// SYNTAX TEST "Step7 AWL.sublime-syntax"

// ==================================================
//  common
//  Performance: 3.0ms
// ==================================================

///////////////////////////////////////////////////////////////////////////////
// namespaces                                                                //
///////////////////////////////////////////////////////////////////////////////

NAMESPACE Name
// <- meta.namespace.plc keyword.declaration.namespace.begin.plc
//^^^^^^^^^^^^^ meta.namespace.plc
//^^^^^^^ keyword.declaration.namespace.begin.plc
//        ^^^^ entity.name.namespace.plc
//            ^ meta.fold.namespace.begin.plc
    TYPE
//  ^^^^^ meta.namespace.plc meta.block.udt.header.plc
//  ^^^^ keyword.declaration.udt.begin.plc
    END_TYPE
//  ^^^^^^^^ meta.namespace.plc keyword.declaration.udt.end.plc

    DATA_BLOCK "dataBlock"
//  ^^^^^^^^^^^^^^^^^^^^^^ meta.namespace.plc meta.block.db.header.plc
//  ^^^^^^^^^^ keyword.declaration.db.begin.plc
//             ^^^^^^^^^^^ entity.name.datablock.plc
//             ^ punctuation.definition.variable.begin.plc
//                       ^ punctuation.definition.variable.end.plc
    END_DATA_BLOCK
//  ^^^^^^^^^^^^^^ meta.namespace.plc keyword.declaration.db.end.plc

    FUNCTION_BLOCK "funcName"
//  ^^^^^^^^^^^^^^^^^^^^^^^^^ meta.namespace.plc meta.block.fb.header.plc
//  ^^^^^^^^^^^^^^ keyword.declaration.fb.begin.plc
//                 ^^^^^^^^^^ entity.name.function.plc
//                 ^ punctuation.definition.variable.begin.plc
//                          ^ punctuation.definition.variable.end.plc
    END_FUNCTION_BLOCK
//  ^^^^^^^^^^^^^^^^^^ meta.namespace.plc keyword.declaration.fb.end.plc

    FUNCTION "funcName"
//  ^^^^^^^^^^^^^^^^^^^ meta.namespace.plc meta.block.fc.header.plc
//  ^^^^^^^^ keyword.declaration.fc.begin.plc
//           ^^^^^^^^^^ entity.name.function.plc
//           ^ punctuation.definition.variable.begin.plc
//                    ^ punctuation.definition.variable.end.plc
    END_FUNCTION
//  ^^^^^^^^^^^^ meta.namespace.plc keyword.declaration.fc.end.plc

    ORGANIZATION_BLOCK "BlockName"
//  ^^^^^^^^^^^^^^^^^^^^^^^^^^^^^^ meta.namespace.plc meta.block.ob.header.plc
//  ^^^^^^^^^^^^^^^^^^ keyword.declaration.ob.begin.plc
//                     ^^^^^^^^^^^ entity.name.organization-block.plc
//                     ^ punctuation.definition.variable.begin.plc
//                               ^ punctuation.definition.variable.end.plc
    END_ORGANIZATION_BLOCK
//  ^^^^^^^^^^^^^^^^^^^^^^ meta.namespace.plc keyword.declaration.ob.end.plc

END_NAMESPACE
// <- meta.namespace.plc keyword.declaration.namespace.end.plc
//^^^^^^^^^^^ meta.namespace.plc keyword.declaration.namespace.end.plc
//           ^ meta.fold.namespace.end.plc - meta.namespace

END_NAMESPACE
// <- invalid.illegal.plc
//^^^^^^^^^^^ invalid.illegal.plc


///////////////////////////////////////////////////////////////////////////////
// datatypes                                                                 //
///////////////////////////////////////////////////////////////////////////////

  TYPE "UDT_TypeName"
//^^^^^^^^^^^^^^^^^^^^ meta.block.udt.header
//^^^^ keyword.declaration.udt.begin
//     ^ punctuation.definition.variable.begin
//     ^^^^^^^^^^^^^^ entity.name.type
//                  ^ punctuation.definition.variable.end
  TITLE = Type Title
//^^^^^^^^^^^^^^^^^^ meta.block.udt.header.plc
//^^^^^^^ meta.mapping.key.plc
//       ^^^^^^^^^^^ meta.mapping.value.plc
//^^^^^ entity.other.attribute-name.title.plc
//      ^ punctuation.separator.key-value.title.plc
//        ^^^^^^^^^^ entity.name.section.plc
   { S7_language := '7(1) Deutsch (Deutschland)  19.01.2014  10:33:55' }
// ^^^^^^^^^^^^^^^^^^^^^^^^^^^^^^^^^^^^^^^^^^^^^^^^^^^^^^^^^^^^^^^^^^^^^ meta.block.udt.header meta.annotation
// ^ punctuation.definition.annotation.begin
//   ^^^^^^^^^^^ variable.annotation
//               ^^ keyword.operator.assignment
//                  ^^^^^^^^^^^^^^^^^^^^^^^^^^^^^^^^^^^^^^^^^^^^^^^^^^ string.quoted.single
//                                                                     ^ punctuation.definition.annotation.end
   NON_RETAIN
// ^^^^^^^^^^ invalid.illegal
   READ_ONLY
// ^^^^^^^^^ invalid.illegal
   VERSION : 1.0
// ^^^^^^^^^^^^^ meta.block.udt.header
// ^^^^^^^^^ meta.mapping.key - meta.mapping.value
//          ^^^^ meta.mapping.value
// ^^^^^^^ entity.other.attribute-name
//         ^ punctuation.separator.key-value
//           ^ constant.numeric.float.version.major
//            ^ punctuation.separator.decimal.version
//             ^ constant.numeric.float.version.minor
   AUTHOR : name
// ^^^^^^^^^^^^^ meta.block.udt.header
// ^^^^^^^^ meta.mapping.key - meta.mapping.value
//         ^^^^^ meta.mapping.value
// ^^^^^^ entity.other.attribute-name
//        ^ punctuation.separator.key-value
//          ^^^^ string.unquoted
   FAMILY : name
// ^^^^^^^^^^^^^ meta.block.udt.header
// ^^^^^^^^ meta.mapping.key - meta.mapping.value
//         ^^^^^ meta.mapping.value
// ^^^^^^ entity.other.attribute-name
//        ^ punctuation.separator.key-value
//          ^^^^ string.unquoted
   NAME : name
// ^^^^^^^^^^^ meta.block.udt.header
// ^^^^^^ meta.mapping.key - meta.mapping.value
//       ^^^^^ meta.mapping.value
// ^^^^ entity.other.attribute-name
//      ^ punctuation.separator.key-value
//        ^^^^ string.unquoted
   ILLEGAL : unknown
// ^^^^^^^^^^^^^^^^^ meta.block.udt.header
// ^^^^^^^ invalid.illegal
//         ^ invalid.illegal
//           ^^^^^^^ invalid.illegal
  STRUCT
//^^^^^^^ meta.block.udt.header meta.struct
//^^^^^^ storage.type.struct.begin
     ID  : INT := 20 ;  //integer
// ^^^^^^^^^^^^^^^^^^^^^^^^^^^^^^^ meta.block.udt.header meta.struct
//   ^^^^^ meta.definition.variable - meta.definition.variable.storage
//        ^^^^^ meta.definition.variable.storage
//             ^^ meta.definition.variable - meta.definition.variable.storage - meta.definition.variable.value
//               ^^^^ meta.definition.variable.value
//   ^^ variable.other
//       ^ punctuation.separator.type
//         ^^^ storage.type.integer
//             ^^ keyword.operator.assignment
//                ^^ meta.number.integer.decimal constant.numeric.value
//                   ^ punctuation.terminator.statement
//                    ^^ - invalid
//                      ^^^^^^^^^ comment.line.double-slash
//                               ^ - invalid
     PTR : POINTER := P#0.0;
// ^^^^^^^^^^^^^^^^^^^^^^^^^^ meta.block.udt.header meta.struct
//   ^^^^^ meta.definition.variable
//        ^^^^^^^^^ meta.definition.variable.storage
//                 ^^ meta.definition.variable
//                   ^^^^^^ meta.definition.variable.value
//   ^^^ variable.other
//       ^ punctuation.separator.type
//         ^^^^^^^ storage.type.pointer
//                 ^^ keyword.operator.assignment
//                    ^^^^^ constant.language.pointer
     TMR : TIMER := T0;
// ^^^^^^^^^^^^^^^^^^^^^ meta.block.udt.header meta.struct
//   ^^^^^ meta.definition.variable
//        ^^^^^^^ meta.definition.variable.storage
//               ^^ meta.definition.variable
//                 ^^^ meta.definition.variable.value
//   ^^^ variable.other
//       ^ punctuation.separator.type
//         ^^^^^ storage.type.timer
//               ^^ keyword.operator.assignment
//                  ^^ variable.language.timer

    //
    // qualified types and variables
    //

    name : _.typeStruct;
//^^^^^^^^^^^^^^^^^^^^^^^ meta.block.udt.header.plc
//  ^^^^^^ meta.definition.variable.plc
//        ^ meta.definition.variable.storage.plc - meta.path
//         ^^^^^^^^^^^^ meta.definition.variable.storage.plc meta.path.plc
//  ^^^^ variable.other.local.plc
//       ^ punctuation.separator.type.plc
//         ^ variable.namespace.plc
//          ^ punctuation.accessor.dot.plc
//           ^^^^^^^^^^ support.type.plc
//                     ^ punctuation.terminator.statement.plc

    name : _.namespace.typeStruct;
//^^^^^^^^^^^^^^^^^^^^^^^^^^^^^^ meta.block.udt.header.plc
//  ^^^^^^ meta.definition.variable.plc
//        ^ meta.definition.variable.storage.plc - meta.path
//         ^^^^^^^^^^^^^^^^^^^^^^ meta.definition.variable.storage.plc meta.path.plc
//  ^^^^ variable.other.local.plc
//       ^ punctuation.separator.type.plc
//         ^ variable.namespace.plc
//          ^ punctuation.accessor.dot.plc
//           ^^^^^^^^^ variable.namespace.plc
//                    ^ punctuation.accessor.dot.plc
//                     ^^^^^^^^^^ support.type.plc
//                               ^ punctuation.terminator.statement.plc

    name : _.name_space_5."type Struct";
//^^^^^^^^^^^^^^^^^^^^^^^^^^^^^^^^^^^^^^ meta.block.udt.header.plc
//  ^^^^^^ meta.definition.variable.plc
//        ^ meta.definition.variable.storage.plc - meta.path
//         ^^^^^^^^^^^^^^^^^^^^^^^^^^^^ meta.definition.variable.storage.plc meta.path.plc
//  ^^^^ variable.other.local.plc
//       ^ punctuation.separator.type.plc
//         ^ variable.namespace.plc
//          ^ punctuation.accessor.dot.plc
//           ^^^^^^^^^^^^ variable.namespace.plc
//                       ^ punctuation.accessor.dot.plc
//                        ^^^^^^^^^^^^^ support.type.plc
//                        ^ punctuation.definition.type.begin.plc
//                                    ^ punctuation.definition.type.end.plc
//                                     ^ punctuation.terminator.statement.plc

    name : Array[1.._.maxItems] of Bool;
//^^^^^^^^^^^^^^^^^^^^^^^^^^^^^^^^^^^^^^ meta.block.udt.header.plc
//  ^^^^^^ meta.definition.variable.plc
//        ^^^^^^^^^^^^^^^^^^^^^^^^^^^^^ meta.definition.variable.storage.plc
//  ^^^^ variable.other.local.plc
//       ^ punctuation.separator.type.plc
//         ^^^^^ storage.type.array.plc
//              ^^^^^^^^^^^^^^^ meta.array-size.plc
//              ^ punctuation.definition.array.begin.plc
//               ^ meta.number.integer.decimal.plc constant.numeric.value.plc
//                ^^ keyword.operator.range.plc
//                  ^^^^^^^^^^ meta.path.plc
//                  ^ variable.namespace.plc
//                   ^ punctuation.accessor.dot.plc
//                    ^^^^^^^^ variable.other.member.plc
//                            ^ punctuation.definition.array.end.plc
//                              ^^ keyword.control.of.plc
//                                 ^^^^ storage.type.bool.plc
//                                     ^ punctuation.terminator.statement.plc

    name : Array[1.._.namespace.maxItems] of Bool;
//^^^^^^^^^^^^^^^^^^^^^^^^^^^^^^^^^^^^^^^^^^^^^^^ meta.block.udt.header.plc
//  ^^^^^^ meta.definition.variable.plc
//        ^^^^^^^^^^^^^^^^^^^^^^^^^^^^^^^^^^^^^^^ meta.definition.variable.storage.plc
//  ^^^^ variable.other.local.plc
//       ^ punctuation.separator.type.plc
//         ^^^^^ storage.type.array.plc
//              ^^^^^^^^^^^^^^^^^^^^^^^^^ meta.array-size.plc
//              ^ punctuation.definition.array.begin.plc
//               ^ meta.number.integer.decimal.plc constant.numeric.value.plc
//                ^^ keyword.operator.range.plc
//                  ^^^^^^^^^^^^^^^^^^^^ meta.path.plc
//                  ^ variable.namespace.plc
//                   ^ punctuation.accessor.dot.plc
//                    ^^^^^^^^^ variable.namespace.plc
//                             ^ punctuation.accessor.dot.plc
//                              ^^^^^^^^ variable.other.member.plc
//                                      ^ punctuation.definition.array.end.plc
//                                        ^^ keyword.control.of.plc
//                                           ^^^^ storage.type.bool.plc
//                                               ^ punctuation.terminator.statement.plc

    _.name : Array[1.._.namespace.datablock.member] of Bool;
//^^^^^^^^^^^^^^^^^^^^^^^^^^^^^^^^^^^^^^^^^^^^^^^^^^^^^^^ meta.block.udt.header.plc
//  ^^^^^^^ meta.definition.variable.plc meta.path.plc
//         ^ meta.definition.variable.plc - meta.path
//          ^^^^^^^^^^^^^^^^^^^^^^^^^^^^^^^^^^^^^^^^^^^^^^^ meta.definition.variable.storage.plc
//  ^ variable.namespace.plc
//   ^ punctuation.accessor.dot.plc
//    ^^^^ variable.other.member.plc
//         ^ punctuation.separator.type.plc
//           ^^^^^ storage.type.array.plc
//                ^^^^^^^^^^^^^^^^^^^^^^^^^^^^^^^^^ meta.array-size.plc
//                ^ punctuation.definition.array.begin.plc
//                 ^ meta.number.integer.decimal.plc constant.numeric.value.plc
//                  ^^ keyword.operator.range.plc
//                    ^^^^^^^^^^^^^^^^^^^^^^^^^^^^ meta.path.plc
//                    ^ variable.namespace.plc
//                     ^ punctuation.accessor.dot.plc
//                      ^^^^^^^^^ variable.namespace.plc
//                               ^ punctuation.accessor.dot.plc
//                                ^^^^^^^^^ variable.namespace.plc
//                                         ^ punctuation.accessor.dot.plc
//                                          ^^^^^^ variable.other.member.plc
//                                                ^ punctuation.definition.array.end.plc
//                                                  ^^ keyword.control.of.plc
//                                                     ^^^^ storage.type.bool.plc
//                                                         ^ punctuation.terminator.statement.plc

  END_STRUCT ;
//^^^^^^^^^^^^^ meta.block.udt.header
//^^^^^^^^^^ meta.struct storage.type.struct.end
//           ^ punctuation.terminator.statement
  BEGIN
//^^^^^^ meta.block.udt.header
//^^^^^ invalid.illegal
  END_TYPE
//^^^^^^^^ meta.block.udt.header
//^^^^^^^^ keyword.declaration.udt.end

///////////////////////////////////////////////////////////////////////////////
// datablocks                                                                //
///////////////////////////////////////////////////////////////////////////////

  DATA_BLOCK "name" // comment
// ^^^^^^^^^^^^^^^^^^^^^^^^^^^ meta.block.db.header
// ^^^^^^^^^ keyword.declaration.db.begin
//           ^ punctuation.definition.variable.begin
//           ^^^^^^ entity.name.datablock
//                ^ punctuation.definition.variable.end
//                  ^^ punctuation.definition.comment.begin
//                  ^^^^^^^^^^ comment.line.double-slash
   TITLE =the datablock description
// ^^^^^^^^^^^^^^^^^^^^^^^^^^^^^^^^ meta.block.db.header
// ^^^^^^^ meta.mapping.key - meta.mapping.value
//        ^^^^^^^^^^^^^^^^^^^^^^^^ meta.mapping.value - meta.mapping.key
// ^^^^^ entity.other.attribute-name.title
//       ^ punctuation.separator.key-value.title
//        ^^^^^^^^^^^^^^^^^^^^^^^^^ entity.name.section
   { S7_language := '7(1) Deutsch (Deutschland)  19.01.2014  10:33:55' }
// ^^^^^^^^^^^^^^^^^^^^^^^^^^^^^^^^^^^^^^^^^^^^^^^^^^^^^^^^^^^^^^^^^^^^^ meta.block.db.header meta.annotation
// ^ punctuation.definition.annotation.begin
//   ^^^^^^^^^^^ variable.annotation
//               ^^ keyword.operator.assignment
//                  ^^^^^^^^^^^^^^^^^^^^^^^^^^^^^^^^^^^^^^^^^^^^^^^^^^ string.quoted.single
//                                                                     ^ punctuation.definition.annotation.end
   NON_RETAIN
// ^^^^^^^^^^ entity.other.attribute-name
   READ_ONLY
// ^^^^^^^^^ entity.other.attribute-name
   VERSION : 1.0
// ^^^^^^^^^^^^^ meta.block.db.header
// ^^^^^^^^^ meta.mapping.key - meta.mapping.value
//          ^^^^ meta.mapping.value
// ^^^^^^^ entity.other.attribute-name
//         ^ punctuation.separator.key-value
//           ^ constant.numeric.float.version.major
//            ^ punctuation.separator.decimal.version
//             ^ constant.numeric.float.version.minor
   AUTHOR : name
// ^^^^^^^^^^^^^ meta.block.db.header
// ^^^^^^^^ meta.mapping.key - meta.mapping.value
//         ^^^^^ meta.mapping.value
// ^^^^^^ entity.other.attribute-name
//        ^ punctuation.separator.key-value
//          ^^^^ string.unquoted
   FAMILY : name
// ^^^^^^^^^^^^^ meta.block.db.header
// ^^^^^^^^ meta.mapping.key - meta.mapping.value
//         ^^^^^ meta.mapping.value
// ^^^^^^ entity.other.attribute-name
//        ^ punctuation.separator.key-value
//          ^^^^ string.unquoted
   NAME : name
// ^^^^^^^^^^^ meta.block.db.header
// ^^^^^^ meta.mapping.key - meta.mapping.value
//       ^^^^^ meta.mapping.value
// ^^^^ entity.other.attribute-name
//      ^ punctuation.separator.key-value
//        ^^^^ string.unquoted
   ILLEGAL : unknown
// ^^^^^^^^^^^^^^^^^ meta.block.db.header
// ^^^^^^^ invalid.illegal
//         ^ invalid.illegal
//           ^^^^^^^ invalid.illegal

   NCK_TypeName
//<- meta.block.db.header
// ^^^^^^^^^^^^^ meta.block.db.header
// ^^^^^^^^^^^^ support.type.plc

   "UDT_TypeName"
//<- meta.block.db.header
// ^^^^^^^^^^^^^^ meta.block.db.header
// ^ punctuation.definition.type.begin
// ^^^^^^^^^^^^^^ support.type.plc
//              ^ punctuation.definition.type.end
   BEGIN illegal // comment
//<- meta.block.db.header
//^ meta.block.db.header - meta.block.db.body
// ^^^^^^^^^^^^^^^^^^^^^^^^ meta.block.db.body - meta.block.db.header
// ^^^^^ keyword.other.begin
//       ^^^^^^^ invalid.illegal
//               ^^ punctuation.definition.comment.begin
//               ^^^^^^^^^^ comment.line.double-slash

   VAR[0].child[ 0 ].attr := W#16#0 ;  // comment
//<- meta.block.db.body
//^^^^^^^^^^^^^^^^^^^^^^^^^^^^^^^^^^^^^^^^^^^^^^^ meta.block.db.body
// ^^^^^^^^^^^^^^^^^^^^^^ meta.path
//    ^^^ meta.brackets
//             ^^^^^ meta.brackets
// ^^^ variable.namespace
//    ^ punctuation.section.brackets.begin
//     ^ meta.number.integer.decimal constant.numeric.value
//      ^ punctuation.section.brackets.end
//       ^ punctuation.accessor.dot
//        ^^^^^ variable.namespace
//             ^ punctuation.section.brackets.begin
//               ^ meta.number.integer.decimal constant.numeric.value
//                 ^ punctuation.section.brackets.end
//                  ^ punctuation.accessor.dot
//                   ^^^^ variable.other.member
//                        ^^ keyword.operator.assignment
//                           ^^^^^^^^^^^^^^^^^^^^^ meta.block.db.body
//                           ^ storage.type.integer
//                            ^ punctuation.separator.type
//                             ^^^ constant.numeric.base
//                               ^ punctuation.separator.base
//                                ^ constant.numeric.value
//                                  ^ punctuation.terminator.statement
   test := W#16 ; illegal // comment
// ^^^^ variable.other.local.plc
//      ^^ keyword.operator.assignment.plc
//         ^^^^ meta.number.integer.decimal.plc
//         ^ storage.type.integer.plc
//          ^ punctuation.separator.type.plc
//           ^^ constant.numeric.value.plc
//              ^ punctuation.terminator.statement.plc
//                ^^^^^^^^ invalid.illegal.eol-expected.plc
//                        ^^^^^^^^^^ comment.line.double-slash.plc
//                        ^^ punctuation.definition.comment.begin.plc

   incomplete
   next_is_valid
// ^^^^^^^^^^^^^ variable.other.local
   date_time := DT#90-1-1-0:0:0.000;
//              ^^^^^^^^^^^^^^^^^^^ meta.number.date-and-time
//              ^^ storage.type.time
//                ^ punctuation.separator.type
//                 ^^^^^^^^^^^^^^^^ constant.numeric.value
//                   ^ punctuation.separator.date
//                     ^ punctuation.separator.date
//                       ^ punctuation.separator.date
//                         ^ punctuation.separator.time
//                           ^ punctuation.separator.time
//                             ^ punctuation.separator.time
   date_time := DT#2017-12-31-23:59:59.999;
//              ^^^^^^^^^^^^^^^^^^^^^^^^^^ meta.number.date-and-time
//              ^^ storage.type.time
//                ^ punctuation.separator.type
//                 ^^^^^^^^^^^^^^^^^^^^^^^ constant.numeric.value
//                     ^ punctuation.separator.date
//                        ^ punctuation.separator.date
//                           ^ punctuation.separator.date
//                              ^ punctuation.separator.time
//                                 ^ punctuation.separator.time
//                                    ^ punctuation.separator.time
   date_time := DT#2017;
//              ^^^^^^^ invalid.illegal
   END_DATA_BLOCK
//<- meta.block.db.body
//^^^^^^^^^^^^^^^ meta.block.db.body
// ^^^^^^^^^^^^^^ keyword.declaration.db.end

DATA_BLOCK "ClassicDB"
   STRUCT
// ^^^^^^ storage.type.struct.begin.plc
      variable : Array[1..5] of "typeVar";
//    ^^^^^^^^^^^^^^^^^^^^^^^^^^^^^^^^^^^ meta.block.db.header.plc meta.struct.plc
//               ^^^^^^^^^^^^^^^^^^^^^^^^ meta.sequence.array.plc
//    ^^^^^^^^ variable.other.local.plc
//             ^ punctuation.separator.type.plc
//               ^^^^^ storage.type.array.plc
//                           ^^ keyword.control.of.plc
//                              ^^^^^^^^^ support.type.plc
//                                       ^ punctuation.terminator.statement.plc
      variable:
            STRUCT
//^^^^^^^^^^^^^^^^^ meta.block.db.header.plc meta.struct.plc meta.definition.variable.storage.plc
//          ^^^^^^^ meta.struct.plc
//          ^^^^^^ storage.type.struct.begin.plc
            END_STRUCT;
//^^^^^^^^^^^^^^^^^^^^ meta.definition.variable.storage.plc meta.struct.plc
//          ^^^^^^^^^^ storage.type.struct.end.plc
//                    ^ punctuation.terminator.statement.plc
   END_STRUCT
// ^^^^^^^^^^ storage.type.struct.end.plc

BEGIN
// <- meta.block.db.body.plc keyword.other.begin.plc
//^^^ meta.block.db.body.plc keyword.other.begin.plc

END_DATA_BLOCK
// <- meta.block.db.body.plc keyword.declaration.db.end.plc
//^^^^^^^^^^^^ meta.block.db.body.plc keyword.declaration.db.end.plc

DATA_BLOCK "TiaDB"
   VAR
// ^^^ keyword.declaration.var.stat.begin.plc
      variable : Array[1..5] of "typeVar";
//    ^^^^^^^^^^^^^^^^^^^^^^^^^^^^^^^^^^^ meta.block.db.header.plc meta.block.var.stat.plc
//               ^^^^^^^^^^^^^^^^^^^^^^^^ meta.sequence.array.plc
//    ^^^^^^^^ variable.other.local.plc
//             ^ punctuation.separator.type.plc
//               ^^^^^ storage.type.array.plc
//                           ^^ keyword.control.of.plc
//                              ^^^^^^^^^ support.type.plc
//                                       ^ punctuation.terminator.statement.plc
   END_VAR
// ^^^^^^^ keyword.declaration.var.end.plc

BEGIN
// <- meta.block.db.body.plc keyword.other.begin.plc
//^^^ meta.block.db.body.plc keyword.other.begin.plc

END_DATA_BLOCK
// <- meta.block.db.body.plc keyword.declaration.db.end.plc
//^^^^^^^^^^^^ meta.block.db.body.plc keyword.declaration.db.end.plc

///////////////////////////////////////////////////////////////////////////////
// functions                                                                 //
///////////////////////////////////////////////////////////////////////////////

   FUNCTION FC 102 : INT  // comment
// ^^^^^^^^^^^^^^^^^^^^^^^^^^^^^^^^^^ meta.block.fc.header
// ^^^^^^^^ keyword.declaration.fc.begin
//          ^^^^^^ entity.name.function
//                 ^ punctuation.separator.mapping.pair
//                   ^^^ storage.type.integer
//                        ^^ punctuation.definition.comment.begin
//                        ^^^^^^^^^^ comment.line.double-slash
   TITLE =the function description
// ^^^^^^^^^^^^^^^^^^^^^^^^^^^^^^^ meta.block.fc.header
// ^^^^^^^ meta.mapping.key - meta.mapping.value
//        ^^^^^^^^^^^^^^^^^^^^^^^^ meta.mapping.value - meta.mapping.key
// ^^^^^ entity.other.attribute-name.title
//       ^ punctuation.separator.key-value.title
//        ^^^^^^^^^^^^^^^^^^^^^^^^ entity.name.section
   { S7_language := '7(1) Deutsch (Deutschland)  19.01.2014  10:33:55' }
// ^^^^^^^^^^^^^^^^^^^^^^^^^^^^^^^^^^^^^^^^^^^^^^^^^^^^^^^^^^^^^^^^^^^^^ meta.block.fc.header meta.annotation
// ^ punctuation.definition.annotation.begin
//   ^^^^^^^^^^^ variable.annotation
//               ^^ keyword.operator.assignment
//                  ^^^^^^^^^^^^^^^^^^^^^^^^^^^^^^^^^^^^^^^^^^^^^^^^^^ string.quoted.single
//                                                                     ^ punctuation.definition.annotation.end
   VERSION : 1.0
// ^^^^^^^^^^^^^ meta.block.fc.header
// ^^^^^^^^^ meta.mapping.key - meta.mapping.value
//          ^^^^ meta.mapping.value
// ^^^^^^^ entity.other.attribute-name
//         ^ punctuation.separator.key-value
//           ^ constant.numeric.float.version.major
//            ^ punctuation.separator.decimal.version
//             ^ constant.numeric.float.version.minor
   AUTHOR : name
// ^^^^^^^^^^^^^ meta.block.fc.header
// ^^^^^^^^ meta.mapping.key - meta.mapping.value
//         ^^^^^ meta.mapping.value
// ^^^^^^ entity.other.attribute-name
//        ^ punctuation.separator.key-value
//          ^^^^ string.unquoted
   FAMILY : name
// ^^^^^^^^^^^^^ meta.block.fc.header
// ^^^^^^^^ meta.mapping.key - meta.mapping.value
//         ^^^^^ meta.mapping.value
// ^^^^^^ entity.other.attribute-name
//        ^ punctuation.separator.key-value
//          ^^^^ string.unquoted
   NAME : name
// ^^^^^^^^^^^ meta.block.fc.header
// ^^^^^^ meta.mapping.key - meta.mapping.value
//       ^^^^^ meta.mapping.value
// ^^^^ entity.other.attribute-name
//      ^ punctuation.separator.key-value
//        ^^^^ string.unquoted
   ILLEGAL : unknown
// ^^^^^^^^^^^^^^^^^ meta.block.fc.header
// ^^^^^^^ invalid.illegal
//         ^ invalid.illegal
//           ^^^^^^^ invalid.illegal

   VAR_INPUT illegal // comment
// <- meta.block.fc.header - meta.block.fc.body
// ^^^^^^^^^^^^^^^^^^^^^^^^^^^^^ meta.block.fc.header meta.block.var.input
// ^^^^^^^^^ keyword.declaration.var.input.begin
//           ^^^^^^^ invalid.illegal.eol-expected
//                   ^^^^^^^^^^ comment.line.double-slash
     RUN : BOOL := TRUE ;  //bool
// ^^^^^^^^^^^^^^^^^^^^^^^^^^^^^^^ meta.block.fc.header meta.block.var.input
//   ^^^^^ meta.definition.variable - meta.definition.variable.storage
//        ^^^^^^ meta.definition.variable.storage - meta.definition.variable.value
//              ^^ meta.definition.variable - meta.definition.variable.storage - meta.definition.variable.value
//                ^^^^^^ meta.definition.variable.value - meta.definition.variable.storage
//   ^^^ variable.other
//       ^ punctuation.separator.type
//         ^^^^ storage.type.bool
//              ^^ keyword.operator.assignment
//                 ^^^^ constant.language.boolean
//                      ^ punctuation.terminator.statement
//                       ^^ - invalid
//                         ^^^^^^ comment.line.double-slash
//                               ^ - invalid
     ID  : INT  ;  //integer
// ^^^^^^^^^^^^^^^^^^^^^^^^^ meta.block.fc.header meta.block.var.input
//   ^^^^^ meta.definition.variable - meta.definition.variable.storage
//        ^^^^^^ meta.definition.variable.storage
//   ^^ variable.other
//       ^ punctuation.separator.type
//         ^^^ storage.type.integer
//              ^ punctuation.terminator.statement
//               ^^ - invalid
//                 ^^^^^^^^^ comment.line.double-slash
//                          ^ - invalid
     _S1  : STRING[32] ;  //string
// ^^^^^^^^^^^^^^^^^^^^^^^^^^^^^^^ meta.block.fc.header meta.block.var.input
//   ^^^^^ meta.definition.variable - meta.definition.variable.storage
//         ^^^^^^^^^^^^ meta.definition.variable.storage
//   ^^^ variable.other
//        ^ punctuation.separator.type
//          ^^^^^^^^^^ storage.type.string
//                     ^ punctuation.terminator.statement
//                      ^^ - invalid
//                        ^^^^^^^^ comment.line.double-slash
//                                ^ - invalid
     _AR  : ARRAY[ 0 .. 20 ] OF //array
// ^^^^^^^^^^^^^^^^^^^^^^^^^^^^^^^^^^^^ meta.block.fc.header meta.block.var.input
//   ^^^^^ meta.definition.variable - meta.definition.variable.storage
//         ^^^^^^^^^^^^^^^^^^^^^^^^^^^^ meta.definition.variable.storage
//          ^^^^^^^^^^^^^^^^^^^^^^^^^^^ meta.sequence.array
//   ^^^ variable.other
//        ^ punctuation.separator.type
//          ^^^^^ storage.type.array
//               ^ punctuation.definition.array.begin
//                 ^ meta.number.integer constant.numeric.value
//                   ^^ keyword.operator.range
//                      ^^ meta.number.integer constant.numeric.value
//                         ^ punctuation.definition.array.end
//                          ^ - invalid
//                           ^^ keyword.control.of
//                             ^ - invalid
//                              ^^ punctuation.definition.comment.begin
//                              ^^^^^^^ comment.line.double-slash
//                                     ^ - invalid
            DWORD := [ DW#16#0, DW#16#2, DW#16#A ] ;  //integer
//^^^^^^^^^^^^^^^^^^^^^^^^^^^^^^^^^^^^^^^^^^^^^^^^^^^^^^^^^^^^^^ meta.block.fc.header meta.block.var.input
//^^^^^^^^^^^^^^^^ meta.definition.variable.storage
//^^^^^^^^^^^^^^^ meta.sequence.array
//               ^^^^ - meta.sequence
//                   ^^^^^^^^^^^^^^^^^^^^^^^^^^^^^ meta.sequence.list
//                                                ^ - meta.sequence
//          ^^^^^ storage.type.integer
//                ^^ keyword.operator.assignment
//                   ^ punctuation.section.sequence.begin
//                     ^^^^^^^ meta.number.integer.hexadecimal
//                            ^ punctuation.separator.sequence
//                              ^^^^^^^ meta.number.integer.hexadecimal
//                                     ^ punctuation.separator.sequence
//                                       ^^^^^^^ meta.number.integer.hexadecimal
//                                               ^ punctuation.section.sequence.end
//                                                ^ - invalid
//                                                 ^ punctuation.terminator.statement
//                                                  ^^ - invalid
//                                                    ^^^^^^^^^ comment.line.double-slash
//                                                             ^ - invalid
     _ST  : STRUCT  //structure
// ^^^^^^^^^^^^^^^^^^^^^^^^^^^^ meta.block.fc.header meta.block.var.input
//   ^^^^^ meta.definition.variable - meta.definition.variable.storage
//         ^^^^^^^^^^^^^^^^^^^^ meta.definition.variable.storage
//          ^^^^^^^^^^^^^^^^^^^ meta.struct
//   ^^^ variable.other
//        ^ punctuation.separator.type
//          ^^^^^^ storage.type.struct.begin
//                  ^^ comment.line.double-slash
//                  ^^^^^^^^^^^ comment.line.double-slash
//                             ^ - invalid
       RUN : BOOL ;  //bool
// ^^^^^^^^^^^^^^^^^^^^^^^^ meta.block.fc.header meta.block.var.input meta.definition.variable.storage meta.struct
//     ^^^^^ meta.definition.variable
//          ^^^^^^ meta.definition.variable.storage meta.definition.variable.storage
//     ^^^ variable.other
//         ^ punctuation.separator.type
//           ^^^^ storage.type.bool
//                ^ punctuation.terminator.statement
//                 ^^ - invalid
//                   ^^^^^^ comment.line.double-slash
//                         ^ - invalid
       ID  : INT  ;  //integer
// ^^^^^^^^^^^^^^^^^^^^^^^^^^^ meta.block.fc.header meta.block.var.input meta.definition.variable.storage meta.struct
//     ^^^^^ meta.definition.variable
//          ^^^^^^ meta.definition.variable.storage meta.definition.variable.storage
//     ^^ variable.other
//         ^ punctuation.separator.type
//           ^^^ storage.type.integer
//                ^ punctuation.terminator.statement
//                 ^^ - invalid
//                   ^^^^^^^^^ comment.line.double-slash
//                            ^ - invalid
       _S1  : STRING[32] := 'initial';  //string
// ^^^^^^^^^^^^^^^^^^^^^^^^^^^^^^^^^^^^^^^^^^^^^^ meta.block.fc.header meta.block.var.input meta.definition.variable.storage meta.struct
//     ^^^^^^ meta.definition.variable
//           ^^^^^^^^^^^^ meta.definition.variable.storage meta.definition.variable.storage
//                       ^^ meta.definition.variable.storage meta.definition.variable
//                         ^^^^^^^^^^ meta.definition.variable.storage meta.definition.variable.value
//     ^^^ variable.other
//          ^ punctuation.separator.type
//            ^^^^^^^^^^ storage.type.string
//                       ^^ keyword.operator.assignment
//                          ^^^^^^^^^ string.quoted.single
//                                   ^ punctuation.terminator.statement
//                                    ^^ - invalid
//                                      ^^^^^^^^ comment.line.double-slash
//                                              ^ - invalid
       _V   : FLOAT := -1.2 ;
// ^^^^^^^^^^^^^^^^^^^^^^^^^^ meta.block.fc.header meta.block.var.input meta.definition.variable.storage meta.struct
//     ^^^^^^ meta.definition.variable
//           ^^^^^^^ meta.definition.variable.storage meta.definition.variable.storage
//                  ^^ meta.definition.variable.storage meta.definition.variable
//                    ^^^^^^ meta.definition.variable.storage meta.definition.variable.value
//     ^^ variable.other
//          ^ punctuation.separator.type
//            ^^^^^ support.type
//                  ^^ keyword.operator.assignment
//                     ^^^^ meta.number.float.decimal
//                     ^ keyword.operator.arithmetic
//                      ^^^ constant.numeric.value
//                       ^ punctuation.separator.decimal
//                          ^ punctuation.terminator.statement
//                           ^^ - invalid
    END_STRUCT ;
// ^^^^^^^^^^^^^ meta.block.fc.header meta.block.var.input
// ^^^^^^^^^^^^ meta.definition.variable.storage
// ^^^^^^^^^^^ meta.struct
//  ^^^^^^^^^^ storage.type.struct.end
//             ^ punctuation.terminator.statement
     _AS  : ARRAY[0..20] OF STRUCT //array
// ^^^^^^^^^^^^^^^^^^^^^^^^^^^^^^^^^^^^^^^^ meta.block.fc.header meta.block.var.input
//   ^^^^^ meta.definition.variable - meta.definition.variable.storage
//         ^^^^^^^^^^^^^^^^^^^^^^^^^^^^^^^ meta.definition.variable.storage
//          ^^^^^^^^^^^^^^^^^^^^^^^^^^^^^^ meta.sequence.array
//                          ^^^^^^^^^^^^^^ meta.struct
//   ^^^ variable.other
//        ^ punctuation.separator.type
//          ^^^^^ storage.type.array
//               ^ punctuation.definition.array.begin
//                ^ meta.number.integer constant.numeric.value
//                 ^^ keyword.operator.range
//                   ^^ meta.number.integer constant.numeric.value
//                     ^ punctuation.definition.array.end
//                       ^^ keyword.control.of
//                          ^^^^^^ storage.type.struct.begin
//                                 ^^ punctuation.definition.comment.begin
//                                 ^^^^^^^ comment.line.double-slash
       RUN : BOOL ;  //bool
// ^^^^^^^^^^^^^^^^^^^^^^^^ meta.block.fc.header meta.block.var.input meta.definition.variable.storage meta.sequence.array meta.struct
//     ^^^^^ meta.definition.variable
//          ^^^^^^ meta.definition.variable.storage meta.definition.variable.storage
//     ^^^ variable.other
//         ^ punctuation.separator.type
//           ^^^^ storage.type.bool
//                ^ punctuation.terminator.statement
//                 ^^ - invalid
//                   ^^^^^^ comment.line.double-slash
//                         ^ - invalid
       ID  : INT  ;  //integer
// ^^^^^^^^^^^^^^^^^^^^^^^^^^^ meta.block.fc.header meta.block.var.input meta.definition.variable.storage meta.sequence.array meta.struct
//     ^^^^^ meta.definition.variable
//          ^^^^^^ meta.definition.variable.storage meta.definition.variable.storage
//     ^^ variable.other
//         ^ punctuation.separator.type
//           ^^^ storage.type.integer
//                ^ punctuation.terminator.statement
//                 ^^ - invalid
//                   ^^^^^^^^^ comment.line.double-slash
//                            ^ - invalid
       _S1  : STRING[32] ;  //string
// ^^^^^^^^^^^^^^^^^^^^^^^^^^^^^^^^^ meta.block.fc.header meta.block.var.input meta.definition.variable.storage meta.sequence.array meta.struct
//     ^^^^^ meta.definition.variable
//           ^^^^^^^^^^^ meta.definition.variable.storage meta.definition.variable.storage
//     ^^^ variable.other
//          ^ punctuation.separator.type
//            ^^^^^^^^^^ storage.type.string
//                       ^ punctuation.terminator.statement
//                        ^^ - invalid
//                          ^^^^^^^^ comment.line.double-slash
//                                  ^ - invalid
    END_STRUCT ;
//^^^^^^^^^^^^^^ meta.block.fc.header meta.block.var.input
//^^^^^^^^^^^^^ meta.definition.variable.storage
//^^^^^^^^^^^^ meta.struct
//  ^^^^^^^^^^ storage.type.struct.end
//             ^ punctuation.terminator.statement
   END_VAR
// <- meta.block.fc.header meta.block.var.input
// ^^^^^^^ meta.block.fc.header meta.block.var.input
// ^^^^^^^ keyword.declaration.var.end

   VAR_OUTPUT
// <- meta.block.fc.header - meta.block.fc.body
// ^^^^^^^^^^ meta.block.fc.header meta.block.var.output
// ^^^^^^^^^^ keyword.declaration.var.output.begin
     RUN : BOOL ;  //bool
// ^^^^^^^^^^^^^^^^^^^^^^ meta.block.fc.header meta.block.var.output
//   ^^^^^ meta.definition.variable - meta.definition.variable.storage
//        ^^^^^^ meta.definition.variable.storage
//   ^^^ variable.other
//       ^ punctuation.separator.type
//         ^^^^ storage.type.bool
//              ^ punctuation.terminator.statement
//               ^^ - invalid
//                 ^^^^^^ comment.line.double-slash
//                       ^ - invalid
     ID  : INT  ;  //integer
// ^^^^^^^^^^^^^^^^^^^^^^^^^ meta.block.fc.header meta.block.var.output
//   ^^^^^ meta.definition.variable - meta.definition.variable.storage
//        ^^^^^^ meta.definition.variable.storage
//   ^^ variable.other
//       ^ punctuation.separator.type
//         ^^^ storage.type.integer
//              ^ punctuation.terminator.statement
//               ^^ - invalid
//                 ^^^^^^^^^ comment.line.double-slash
//                          ^ - invalid
     _S1  : STRING[32] ;  //string
// ^^^^^^^^^^^^^^^^^^^^^^^^^^^^^^^ meta.block.fc.header meta.block.var.output
//   ^^^^^ meta.definition.variable - meta.definition.variable.storage
//         ^^^^^^^^^^^^ meta.definition.variable.storage
//   ^^^ variable.other
//        ^ punctuation.separator.type
//          ^^^^^^^^^^ storage.type.string
//                     ^ punctuation.terminator.statement
//                      ^^ - invalid
//                        ^^^^^^^^ comment.line.double-slash
//                                ^ - invalid
     _AR  : ARRAY[ 0 .. 20 ] OF //array
// ^^^^^^^^^^^^^^^^^^^^^^^^^^^^^^^^^^^^ meta.block.fc.header meta.block.var.output
//   ^^^^^ meta.definition.variable - meta.definition.variable.storage
//         ^^^^^^^^^^^^^^^^^^^^^^^^^^^^ meta.definition.variable.storage
//          ^^^^^^^^^^^^^^^^^^^^^^^^^^^ meta.sequence.array
//   ^^^ variable.other
//        ^ punctuation.separator.type
//          ^^^^^ storage.type.array
//               ^ punctuation.definition.array.begin
//                 ^ meta.number.integer constant.numeric.value
//                   ^^ keyword.operator.range
//                      ^^ meta.number.integer constant.numeric.value
//                         ^ punctuation.definition.array.end
//                           ^^ keyword.control.of
//                              ^^ punctuation.definition.comment.begin
//                              ^^^^^^^ comment.line.double-slash
            DWORD ;  //integer
// ^^^^^^^^^^^^^^^^^^^^^^^^^^^ meta.block.fc.header meta.block.var.output
// ^^^^^^^^^^^^^^ meta.definition.variable.storage meta.sequence.array
//          ^^^^^ storage.type.integer
//                   ^^^^^^^^^ comment.line.double-slash
//                            ^ - invalid
     _ST  : STRUCT  //structure
// ^^^^^^^^^^^^^^^^^^^^^^^^^^^^ meta.block.fc.header meta.block.var.output
//   ^^^^^ meta.definition.variable - meta.definition.variable.storage
//         ^^^^^^^^^^^^^^^^^^^^ meta.definition.variable.storage
//          ^^^^^^^^^^^^^^^^^^^ meta.struct
//   ^^^ variable.other
//        ^ punctuation.separator.type
//          ^^^^^^ storage.type.struct.begin
//                  ^^^^^^^^^^^ comment.line.double-slash
//                             ^ - invalid
       RUN : BOOL ;  //bool
// ^^^^^^^^^^^^^^^^^^^^^^^^ meta.block.fc.header meta.block.var.output meta.definition.variable.storage meta.struct
//     ^^^^^ meta.definition.variable
//          ^^^^^^ meta.definition.variable.storage meta.definition.variable.storage
//     ^^^ variable.other
//         ^ punctuation.separator.type
//           ^^^^ storage.type.bool
//                ^ punctuation.terminator.statement
//                   ^^^^^^ comment.line.double-slash
//                         ^ - invalid
       ID  : INT  ;  //integer
// ^^^^^^^^^^^^^^^^^^^^^^^^^^^ meta.block.fc.header meta.block.var.output meta.definition.variable.storage meta.struct
//     ^^^^^ meta.definition.variable
//          ^^^^^^ meta.definition.variable.storage meta.definition.variable.storage
//     ^^ variable.other
//         ^ punctuation.separator.type
//           ^^^ storage.type.integer
       _S1  : STRING[32] ;  //string
// ^^^^^^^^^^^^^^^^^^^^^^^^^^^^^^^^^ meta.block.fc.header meta.block.var.output meta.definition.variable.storage meta.struct
//     ^^^^^ meta.definition.variable
//           ^^^^^^^^^^^ meta.definition.variable.storage meta.definition.variable.storage
//     ^^^ variable.other
//          ^ punctuation.separator.type
//            ^^^^^^^^^^ storage.type.string
    END_STRUCT ;
//^^^^^^^^^^^^^^^ meta.block.fc.header meta.block.var.output
//^^^^^^^^^^^^^ meta.definition.variable.storage
//^^^^^^^^^^^^ meta.struct
//  ^^^^^^^^^^ storage.type.struct.end
//             ^ punctuation.terminator.statement
//              ^ - invalid
     _AS  : ARRAY[ 0 .. 20 ] OF STRUCT //array
// ^^^^^^^^^^^^^^^^^^^^^^^^^^^^^^^^^^^^^^^^^^^ meta.block.fc.header meta.block.var.output
//   ^^^^^ meta.definition.variable - meta.definition.variable.storage
//         ^^^^^^^^^^^^^^^^^^^^^^^^^^^^^^^^^^^ meta.definition.variable.storage
//          ^^^^^^^^^^^^^^^^^^^^^^^^^^^^^^^^^^ meta.sequence.array
//                              ^^^^^^^^^^^^^^ meta.struct
//   ^^^ variable.other
//        ^ punctuation.separator.type
//          ^^^^^ storage.type.array
//               ^ punctuation.definition.array.begin
//                 ^ meta.number.integer constant.numeric.value
//                   ^^ keyword.operator.range
//                      ^^ meta.number.integer constant.numeric.value
//                         ^ punctuation.definition.array.end
//                           ^^ keyword.control.of
//                              ^^^^^^ storage.type.struct.begin
//                                     ^^ punctuation.definition.comment.begin
//                                     ^^^^^^^ comment.line.double-slash
//                                            ^ - invalid
       RUN : BOOL ;  //bool
// ^^^^^^^^^^^^^^^^^^^^^^^^ meta.block.fc.header meta.block.var.output meta.definition.variable.storage meta.sequence.array meta.struct
//     ^^^^^ meta.definition.variable
//          ^^^^^^ meta.definition.variable.storage meta.definition.variable.storage
//     ^^^ variable.other
//         ^ punctuation.separator.type
//           ^^^^ storage.type.bool
       ID  : INT  ;  //integer
// ^^^^^^^^^^^^^^^^^^^^^^^^^^^ meta.block.fc.header meta.block.var.output meta.definition.variable.storage meta.sequence.array meta.struct
//     ^^^^^ meta.definition.variable
//          ^^^^^^ meta.definition.variable.storage meta.definition.variable.storage
//     ^^ variable.other
//         ^ punctuation.separator.type
//           ^^^ storage.type.integer
       _S1  : STRING[32] ;  //string
// ^^^^^^^^^^^^^^^^^^^^^^^^^^^^^^^^^ meta.block.fc.header meta.block.var.output meta.definition.variable.storage meta.sequence.array meta.struct
//     ^^^^^ meta.definition.variable
//           ^^^^^^^^^^^ meta.definition.variable.storage meta.definition.variable.storage
//     ^^^ variable.other
//          ^ punctuation.separator.type
//            ^^^^^^^^^^ storage.type.string
    END_STRUCT ;
//^^^^^^^^^^^^^^^ meta.block.fc.header meta.block.var
//^^^^^^^^^^^^^ meta.definition.variable.storage
//^^^^^^^^^^^^ meta.struct
//  ^^^^^^^^^^ storage.type.struct.end
//             ^ punctuation.terminator.statement
//              ^ - invalid
   END_VAR
// <- meta.block.fc.header meta.block.var.output
// ^^^^^^^ meta.block.fc.header meta.block.var.output
// ^^^^^^^ keyword.declaration.var.end

   VAR_IN_OUT
// <- meta.block.fc.header - meta.block.fc.body
// ^^^^^^^^^^ meta.block.fc.header meta.block.var.in-out
// ^^^^^^^^^^ keyword.declaration.var.in-out.begin
     RUN : BOOL ;  //bool
// ^^^^^^^^^^^^^^^^^^^^^^ meta.block.fc.header meta.block.var.in-out
//   ^^^^^ meta.definition.variable - meta.definition.variable.storage
//        ^^^^^^ meta.definition.variable.storage
//   ^^^ variable.other
//       ^ punctuation.separator.type
//         ^^^^ storage.type.bool
     ID  : INT  ;  //integer
// ^^^^^^^^^^^^^^^^^^^^^^^^^ meta.block.fc.header meta.block.var.in-out
//   ^^^^^ meta.definition.variable - meta.definition.variable.storage
//        ^^^^^^ meta.definition.variable.storage
//   ^^ variable.other
//       ^ punctuation.separator.type
//         ^^^ storage.type.integer
     _S1  : STRING[32] ;  //string
// ^^^^^^^^^^^^^^^^^^^^^^^^^^^^^^^ meta.block.fc.header meta.block.var.in-out
//   ^^^^^ meta.definition.variable - meta.definition.variable.storage
//         ^^^^^^^^^^^^ meta.definition.variable.storage
//   ^^^ variable.other
//        ^ punctuation.separator.type
//          ^^^^^^^^^^ storage.type.string
     _AR  : ARRAY[ 0 .. 20 ] OF //array
// ^^^^^^^^^^^^^^^^^^^^^^^^^^^^^^^^^^^^ meta.block.fc.header meta.block.var.in-out
//   ^^^^^ meta.definition.variable - meta.definition.variable.storage
//         ^^^^^^^^^^^^^^^^^^^^^^^^^^^^ meta.definition.variable.storage
//          ^^^^^^^^^^^^^^^^^^^^^^^^^^^ meta.sequence.array
//   ^^^ variable.other
//        ^ punctuation.separator.type
//          ^^^^^ storage.type.array
//               ^ punctuation.definition.array.begin
//                 ^ meta.number.integer constant.numeric.value
//                   ^^ keyword.operator.range
//                      ^^ meta.number.integer constant.numeric.value
//                         ^ punctuation.definition.array.end
//                           ^^ keyword.control.of
//                              ^^ punctuation.definition.comment.begin
//                              ^^^^^^^ comment.line.double-slash
            DWORD ;  //integer
// ^^^^^^^^^^^^^^^^^^^^^^^^^^^ meta.block.fc.header meta.block.var.in-out
// ^^^^^^^^^^^^^^ meta.definition.variable.storage meta.sequence.array
//          ^^^^^ storage.type.integer
     _ST  : STRUCT  //structure
// ^^^^^^^^^^^^^^^^^^^^^^^^^^^^ meta.block.fc.header meta.block.var.in-out
//   ^^^^^ meta.definition.variable - meta.definition.variable.storage
//         ^^^^^^^^^^^^^^^^^^^^ meta.definition.variable.storage
//          ^^^^^^^^^^^^^^^^^^^ meta.struct
//   ^^^ variable.other
//        ^ punctuation.separator.type
//          ^^^^^^ storage.type.struct.begin
       RUN : BOOL ;  //bool
// ^^^^^^^^^^^^^^^^^^^^^^^^ meta.block.fc.header meta.block.var.in-out meta.definition.variable.storage meta.struct
//     ^^^^^ meta.definition.variable
//          ^^^^^^ meta.definition.variable.storage meta.definition.variable.storage
//     ^^^ variable.other
//         ^ punctuation.separator.type
//           ^^^^ storage.type.bool
       ID  : INT  ;  //integer
// ^^^^^^^^^^^^^^^^^^^^^^^^^^^ meta.block.fc.header meta.block.var.in-out meta.definition.variable.storage meta.struct
//     ^^^^^ meta.definition.variable
//          ^^^^^^ meta.definition.variable.storage meta.definition.variable.storage
//     ^^ variable.other
//         ^ punctuation.separator.type
//           ^^^ storage.type.integer
       _S1  : STRING[32] ;  //string
// ^^^^^^^^^^^^^^^^^^^^^^^^^^^^^^^^^ meta.block.fc.header meta.block.var.in-out meta.definition.variable.storage meta.struct
//     ^^^^^ meta.definition.variable
//           ^^^^^^^^^^^ meta.definition.variable.storage meta.definition.variable.storage
//     ^^^ variable.other
//          ^ punctuation.separator.type
//            ^^^^^^^^^^ storage.type.string
    END_STRUCT ;
//^^^^^^^^^^^^^^^ meta.block.fc.header meta.block.var.in-out
//^^^^^^^^^^^^^ meta.definition.variable.storage
//^^^^^^^^^^^^ meta.struct
//  ^^^^^^^^^^ storage.type.struct.end
//             ^ punctuation.terminator.statement
//              ^ - invalid
     _AS  : ARRAY[ 0 .. 20 ] OF STRUCT //array
// ^^^^^^^^^^^^^^^^^^^^^^^^^^^^^^^^^^^^^^^^^^^ meta.block.fc.header meta.block.var.in-out
//   ^^^^^ meta.definition.variable - meta.definition.variable.storage
//         ^^^^^^^^^^^^^^^^^^^^^^^^^^^^^^^^^^^ meta.definition.variable.storage
//          ^^^^^^^^^^^^^^^^^^^^^^^^^^^^^^^^^^ meta.sequence.array
//                              ^^^^^^^^^^^^^^ meta.struct
//   ^^^ variable.other
//        ^ punctuation.separator.type
//          ^^^^^ storage.type.array
//               ^ punctuation.definition.array.begin
//                 ^ meta.number.integer constant.numeric.value
//                   ^^ keyword.operator.range
//                      ^^ meta.number.integer constant.numeric.value
//                         ^ punctuation.definition.array.end
//                           ^^ keyword.control.of
//                              ^^^^^^ storage.type.struct.begin
//                                     ^^ punctuation.definition.comment.begin
//                                     ^^^^^^^ comment.line.double-slash
       RUN : BOOL ;  //bool
// ^^^^^^^^^^^^^^^^^^^^^^^^ meta.block.fc.header meta.block.var.in-out meta.definition.variable.storage meta.sequence.array meta.struct
//     ^^^^^ meta.definition.variable
//          ^^^^^^ meta.definition.variable.storage meta.definition.variable.storage
//     ^^^ variable.other
//         ^ punctuation.separator.type
//           ^^^^ storage.type.bool
       ID  : INT  ;  //integer
// ^^^^^^^^^^^^^^^^^^^^^^^^^^^ meta.block.fc.header meta.block.var.in-out meta.definition.variable.storage meta.sequence.array meta.struct
//     ^^^^^ meta.definition.variable
//          ^^^^^^ meta.definition.variable.storage meta.definition.variable.storage
//     ^^ variable.other
//         ^ punctuation.separator.type
//           ^^^ storage.type.integer
       _S1  : STRING[32] ;  //string
// ^^^^^^^^^^^^^^^^^^^^^^^^^^^^^^^^^ meta.block.fc.header meta.block.var.in-out meta.definition.variable.storage meta.sequence.array meta.struct
//     ^^^^^ meta.definition.variable
//           ^^^^^^^^^^^^ meta.definition.variable.storage meta.definition.variable.storage
//     ^^^ variable.other
//          ^ punctuation.separator.type
//            ^^^^^^^^^^ storage.type.string
    END_STRUCT ;
//^^^^^^^^^^^^^^^ meta.block.fc.header meta.block.var.in-out
//^^^^^^^^^^^^^ meta.definition.variable.storage
//^^^^^^^^^^^^ meta.struct
//  ^^^^^^^^^^ storage.type.struct.end
//             ^ punctuation.terminator.statement
    "name" : String;   // program name
//^^^^^^^^^^^^^^^^^^^ meta.block.fc.header meta.block.var.in-out
//  ^^^^^^^ meta.definition.variable.plc
//  ^^^^^^ variable.other.local.plc
//         ^ punctuation.separator.type.plc
//           ^^^^^^ storage.type.string.plc
//                 ^ punctuation.terminator.statement.plc
   END_VAR
// <- meta.block.fc.header meta.block.var.in-out
// ^^^^^^^ meta.block.fc.header meta.block.var.in-out
// ^^^^^^^ keyword.declaration.var.end

   VAR_TEMP
// <- meta.block.fc.header - meta.block.fc.body
// ^^^^^^^^ meta.block.fc.header meta.block.var.temp
// ^^^^^^^^ keyword.declaration.var.temp.begin
     RUN : BOOL ;  //bool
// ^^^^^^^^^^^^^^^^^^^^^^ meta.block.fc.header meta.block.var.temp
//   ^^^^^ meta.definition.variable - meta.definition.variable.storage
//        ^^^^^^ meta.definition.variable.storage
//   ^^^ variable.other
//       ^ punctuation.separator.type
//         ^^^^ storage.type.bool
     ID  : INT  ;  //integer
// ^^^^^^^^^^^^^^^^^^^^^^^^^ meta.block.fc.header meta.block.var.temp
//   ^^^^^ meta.definition.variable - meta.definition.variable.storage
//        ^^^^^^ meta.definition.variable.storage
//   ^^ variable.other
//       ^ punctuation.separator.type
//         ^^^ storage.type.integer
     _S1  : STRING[32] ;  //string
// ^^^^^^^^^^^^^^^^^^^^^^^^^^^^^^^ meta.block.fc.header meta.block.var.temp
//   ^^^^^ meta.definition.variable - meta.definition.variable.storage
//         ^^^^^^^^^^^^ meta.definition.variable.storage
//   ^^^ variable.other
//        ^ punctuation.separator.type
//          ^^^^^^^^^^ storage.type.string
     _AR  : ARRAY[ 0 .. 20 ] OF //array
// ^^^^^^^^^^^^^^^^^^^^^^^^^^^^^^^^^^^^ meta.block.fc.header meta.block.var.temp
//   ^^^^^ meta.definition.variable - meta.definition.variable.storage
//         ^^^^^^^^^^^^^^^^^^^^^^^^^^^^ meta.definition.variable.storage
//          ^^^^^^^^^^^^^^^^^^^^^^^^^^^ meta.sequence.array
//   ^^^ variable.other
//        ^ punctuation.separator.type
//          ^^^^^ storage.type.array
//               ^ punctuation.definition.array.begin
//                 ^ meta.number.integer constant.numeric.value
//                   ^^ keyword.operator.range
//                      ^^ meta.number.integer constant.numeric.value
//                         ^ punctuation.definition.array.end
//                           ^^ keyword.control.of
//                              ^^ punctuation.definition.comment.begin
//                              ^^^^^^^ comment.line.double-slash
            DWORD ;  //integer
// ^^^^^^^^^^^^^^^^^^^^^^^^^^^ meta.block.fc.header meta.block.var.temp
// ^^^^^^^^^^^^^^ meta.definition.variable.storage meta.sequence.array
//          ^^^^^ storage.type.integer
     _ST  : STRUCT  //structure
// ^^^^^^^^^^^^^^^^^^^^^^^^^^^^ meta.block.fc.header meta.block.var.temp
//   ^^^^^ meta.definition.variable - meta.definition.variable.storage
//         ^^^^^^^^^^^^^^^^^^^^ meta.definition.variable.storage
//          ^^^^^^^^^^^^^^^^^^^ meta.struct
//   ^^^ variable.other
//        ^ punctuation.separator.type
//          ^^^^^^ storage.type.struct.begin
       RUN : BOOL ;  //bool
// ^^^^^^^^^^^^^^^^^^^^^^^^ meta.block.fc.header meta.block.var.temp meta.definition.variable.storage meta.struct
//     ^^^^^ meta.definition.variable
//          ^^^^^^ meta.definition.variable.storage meta.definition.variable.storage
//     ^^^ variable.other
//         ^ punctuation.separator.type
//           ^^^^ storage.type.bool
       ID  : INT  ;  //integer
// ^^^^^^^^^^^^^^^^^^^^^^^^^^^ meta.block.fc.header meta.block.var.temp meta.definition.variable.storage meta.struct
//     ^^^^^ meta.definition.variable
//          ^^^^^^ meta.definition.variable.storage meta.definition.variable.storage
//     ^^ variable.other
//         ^ punctuation.separator.type
//           ^^^ storage.type.integer
       _S1  : STRING[32] ;  //string
// ^^^^^^^^^^^^^^^^^^^^^^^^^^^^^^^^^ meta.block.fc.header meta.block.var.temp meta.definition.variable.storage meta.struct
//     ^^^^^ meta.definition.variable
//           ^^^^^^^^^^^^ meta.definition.variable.storage meta.definition.variable.storage
//     ^^^ variable.other
//          ^ punctuation.separator.type
//            ^^^^^^^^^^ storage.type.string
    END_STRUCT ;
//^^^^^^^^^^^^^^^ meta.block.fc.header meta.block.var.temp
//^^^^^^^^^^^^^ meta.definition.variable.storage
//^^^^^^^^^^^^ meta.struct
//  ^^^^^^^^^^ storage.type.struct.end
//             ^ punctuation.terminator.statement
     _AS  : ARRAY[ 0 .. 20 ] OF STRUCT //array
// ^^^^^^^^^^^^^^^^^^^^^^^^^^^^^^^^^^^^^^^^^^^ meta.block.fc.header meta.block.var.temp
//   ^^^^^ meta.definition.variable - meta.definition.variable.storage
//         ^^^^^^^^^^^^^^^^^^^^^^^^^^^^^^^^^^^ meta.definition.variable.storage
//          ^^^^^^^^^^^^^^^^^^^^^^^^^^^^^^^^^^ meta.sequence.array
//                              ^^^^^^^^^^^^^^ meta.struct
//   ^^^ variable.other
//        ^ punctuation.separator.type
//          ^^^^^ storage.type.array
//               ^ punctuation.definition.array.begin
//                 ^ meta.number.integer constant.numeric.value
//                   ^^ keyword.operator.range
//                      ^^ meta.number.integer constant.numeric.value
//                         ^ punctuation.definition.array.end
//                           ^^ keyword.control.of
//                              ^^^^^^ storage.type.struct.begin
//                                     ^^ punctuation.definition.comment.begin
//                                     ^^^^^^^ comment.line.double-slash
       RUN : BOOL ;  //bool
// ^^^^^^^^^^^^^^^^^^^^^^^^ meta.block.fc.header meta.block.var.temp meta.definition.variable.storage meta.sequence.array meta.struct
//     ^^^^^ meta.definition.variable
//          ^^^^^^ meta.definition.variable.storage meta.definition.variable.storage
//     ^^^ variable.other
//         ^ punctuation.separator.type
//           ^^^^ storage.type.bool
       ID  : INT  ;  //integer
// ^^^^^^^^^^^^^^^^^^^^^^^^^^^ meta.block.fc.header meta.block.var.temp meta.definition.variable.storage meta.sequence.array meta.struct
//     ^^^^^ meta.definition.variable
//          ^^^^^^ meta.definition.variable.storage meta.definition.variable.storage
//     ^^ variable.other
//         ^ punctuation.separator.type
//           ^^^ storage.type.integer
       _S1  : STRING[32] ;  //string
// ^^^^^^^^^^^^^^^^^^^^^^^^^^^^^^^^^ meta.block.fc.header meta.block.var.temp meta.definition.variable.storage meta.sequence.array meta.struct
//     ^^^^^ meta.definition.variable
//           ^^^^^^^^^^^^ meta.definition.variable.storage meta.definition.variable.storage
//     ^^^ variable.other
//          ^ punctuation.separator.type
//            ^^^^^^^^^^ storage.type.string
    END_STRUCT ;
//^^^^^^^^^^^^^^^ meta.block.fc.header meta.block.var.temp
//^^^^^^^^^^^^^ meta.definition.variable.storage
//^^^^^^^^^^^^ meta.struct
//  ^^^^^^^^^^ storage.type.struct.end
//             ^ punctuation.terminator.statement
   END_VAR
// <- meta.block.fc.header meta.block.var.temp
// ^^^^^^^ meta.block.fc.header meta.block.var.temp
// ^^^^^^^ keyword.declaration.var.end

   VAR CONSTANT
//^^^^^^^^^^^^^ meta.block.fc.header.plc
// ^^^^^^^^^^^^ meta.block.var.constant.plc keyword.declaration.var.constant.begin.plc
   END_VAR
// <- meta.block.fc.header.plc meta.block.var.constant.plc
//^^^^^^^^ meta.block.fc.header.plc meta.block.var.constant.plc
// ^^^^^^^ keyword.declaration.var.end.plc

   VAR
// ^^^ meta.block.fc.header invalid.illegal
   END_VAR
// ^^^^^^^ meta.block.fc.header invalid.illegal

// NOTE: unclosed input declaration context

   VAR_INPUT
// ^^^^^^^^^ keyword.declaration.var.input.begin

   BEGIN
// <- meta.block.fc.header - meta.block.fc.body
//^ meta.block.fc.header - meta.block.fc.body
// ^^^^^ meta.block.fc.body - meta.block.fc.header
// ^^^^^ keyword.other.begin

   NETWORK //network 1
// <- meta.block.fc.body
// ^^^^^^^^^^^^^^^^^^^ meta.block.fc.body meta.block.network
// ^^^^^^^ keyword.control.network
   TITLE =CALL test
// <- meta.block.fc.body meta.block.network
// ^^^^^^^^^^^^^^^^ meta.block.fc.body meta.block.network
// ^^^^^^^ meta.mapping.key
//        ^^^^^^^^^ meta.mapping.value
// ^^^^^ entity.other.attribute-name.title
//       ^ punctuation.separator.key-value.title
//        ^^^^^^^^^ entity.name.section

///////////////////////////////////////////////////////////////////////////////
// basic operations                                                          //
///////////////////////////////////////////////////////////////////////////////

      BLD  1; // comment
//    ^^^ keyword.operator.nop
//         ^ meta.number.integer constant.numeric.value
//          ^ punctuation.terminator.statement
      NOP  0; // comment
//    ^^^ keyword.operator.nop
//         ^ meta.number.integer constant.numeric.value
//          ^ punctuation.terminator.statement

///////////////////////////////////////////////////////////////////////////////
// datablock operations                                                      //
///////////////////////////////////////////////////////////////////////////////

      AUF   DB 10;
// <- meta.block.fc.body meta.block.network
//^^^^^^^^^^^^^^^^^ meta.block.fc.body meta.block.network
//       ^^^^^^^^ meta.operand.datablock
//               ^^ - meta.operand.datablock
//    ^^^ keyword.operator.load.db
//          ^^^^^ variable.language.db
//               ^ punctuation.terminator.statement
      AUF   DB [MW 10];
// <- meta.block.fc.body meta.block.network
//^^^^^^^^^^^^^^^^^^^^^ meta.block.fc.body meta.block.network
//       ^^^ meta.operand.datablock - meta.address
//          ^^^ meta.operand.datablock meta.address.indirect - meta.brackets
//             ^^^^^^^ meta.operand.datablock meta.address.indirect meta.brackets
//                    ^^ - meta.operand.datablock
//    ^^^ keyword.operator.load.db
//          ^^^^^^^^^^ meta.address.indirect
//          ^^ variable.language.timer
//             ^ punctuation.section.brackets.begin
//              ^^^^^ variable.language.address
//                   ^ punctuation.section.brackets.end
//                    ^ punctuation.terminator.statement
      AUF   "IDB_Block";
// <- meta.block.fc.body meta.block.network
//^^^^^^^^^^^^^^^^^^^^^^^ meta.block.fc.body meta.block.network
//       ^^^^^^^^^^^^^^ meta.operand.datablock
//                     ^^ - meta.operand.datablock
//    ^^^ keyword.operator.load.db
//          ^^^^^^^^^^^ variable.other.global
//          ^ punctuation.definition.variable.begin
//                    ^ punctuation.definition.variable.end
//                     ^ punctuation.terminator.statement
      AUF   DBNO;
// <- meta.block.fc.body meta.block.network
//^^^^^^^^^^^^^^^^ meta.block.fc.body meta.block.network
//       ^^^^^^^ meta.operand.datablock
//              ^^ - meta.operand.datablock
//    ^^^ keyword.operator.load.db
//          ^^^^ invalid.illegal
//              ^ punctuation.terminator.statement
      AUF   DINO;
// <- meta.block.fc.body meta.block.network
//^^^^^^^^^^^^^^^^ meta.block.fc.body meta.block.network
//       ^^^^^^^ meta.operand.datablock
//              ^^ - meta.operand.datablock
//    ^^^ keyword.operator.load.db
//          ^^^^ invalid.illegal
//              ^ punctuation.terminator.statement
      TDB   ;
// <- meta.block.fc.body meta.block.network
//^^^^^^^^^^^^^^^^ meta.block.fc.body meta.block.network
//    ^^^ keyword.operator.db
//          ^ punctuation.terminator.statement

///////////////////////////////////////////////////////////////////////////////
// logical operations                                                        //
///////////////////////////////////////////////////////////////////////////////

      U     E3.0;
// <- meta.block.fc.body meta.block.network
// ^^^^^^^^^^^^^^^ meta.block.fc.body meta.block.network
//     ^^^^^^^^^ meta.operand.logical
//              ^^ - meta.operand
//    ^ keyword.operator.logical
//          ^^^^ variable.language.address
//            ^ punctuation.separator.decimal
//              ^ punctuation.terminator.statement
//               ^ - invalid
      U     A3.0;
// <- meta.block.fc.body meta.block.network
// ^^^^^^^^^^^^^^^ meta.block.fc.body meta.block.network
//     ^^^^^^^^^ meta.operand.logical
//              ^^ - meta.operand
//    ^ keyword.operator.logical
//          ^^^^ variable.language.address
//            ^ punctuation.separator.decimal
//              ^ punctuation.terminator.statement
//               ^ - invalid
      U     L3.0;
// <- meta.block.fc.body meta.block.network
// ^^^^^^^^^^^^^^^ meta.block.fc.body meta.block.network
//     ^^^^^^^^^ meta.operand.logical
//              ^^ - meta.operand
//    ^ keyword.operator.logical
//          ^^^^ variable.language.address
//            ^ punctuation.separator.decimal
//              ^ punctuation.terminator.statement
//               ^ - invalid
      U     M3.0;
// <- meta.block.fc.body meta.block.network
// ^^^^^^^^^^^^^^^ meta.block.fc.body meta.block.network
//     ^^^^^^^^^ meta.operand.logical
//              ^^ - meta.operand
//    ^ keyword.operator.logical
//          ^^^^ variable.language.address
//            ^ punctuation.separator.decimal
//              ^ punctuation.terminator.statement
//               ^ - invalid
      U     DBX3.0;
// <- meta.block.fc.body meta.block.network
// ^^^^^^^^^^^^^^^^^ meta.block.fc.body meta.block.network
//     ^^^^^^^^^^^ meta.operand.logical
//                ^^ - meta.operand
//    ^ keyword.operator.logical
//          ^^^^^^ variable.language.address
//              ^ punctuation.separator.decimal
//                ^ punctuation.terminator.statement
//                 ^ - invalid
      U     DIX3.0;
// <- meta.block.fc.body meta.block.network
// ^^^^^^^^^^^^^^^^^ meta.block.fc.body meta.block.network
//     ^^^^^^^^^^^ meta.operand.logical
//                ^^ - meta.operand
//    ^ keyword.operator.logical
//          ^^^^^^ variable.language.address
//              ^ punctuation.separator.decimal
//                ^ punctuation.terminator.statement
//                 ^ - invalid
      U     DB10.DBX3.0;
// <- meta.block.fc.body meta.block.network
// ^^^^^^^^^^^^^^^^^^^^^^ meta.block.fc.body meta.block.network
//     ^^^^^^^^^^^^^^^^ meta.operand.logical
//                     ^^ - meta.operand
//    ^ keyword.operator.logical
//          ^^^^ variable.language.db
//              ^ punctuation.accessor.dot
//               ^^^^^^ variable.language.address
//                   ^ punctuation.separator.decimal
//                     ^ punctuation.terminator.statement
//                      ^ - invalid

